FUNCTION_BLOCK FB_LogCounterValue IMPLEMENTS I_VisitModules
VAR_INPUT
END_VAR
VAR_OUTPUT
END_VAR
VAR
END_VAR

METHOD VisitModules
VAR_INPUT
	Module	: I_Module;
END_VAR
ADSLOGDINT(ADSLOG_MSGTYPE_HINT OR ADSLOG_MSGTYPE_LOG, 'The Module Counter is: %d', Module.CounterValue);
END_METHOD

END_FUNCTION_BLOCK

(* stored: Version 1.1.0.1, ProductVersion 3.1.4024.12
   POU FB_LogCounterValue: Id {f760fbc9-0e16-4a7b-bf35-36e8de23677b}, SpecialFunc None
   Method VisitModules: Id {af05c526-8211-4af5-8a6a-99c1cbfc2c78} *)
